Yaskawa INFORM job: CHECKWEAVEADJUSTVALUE.JBI

/JOB
//NAME CHECKWEAVEADJUSTVALUE
//POS
///NPOS 0,0,0,0,0,0
//INST
///DATE 2025/09/26 10:45
///ATTR SC,RW
///GROUP1 RB1
NOP
WVADJ STD=65.536 ST=65.536 END=65.536 LEN=65.536 ADJMD=0
END
